INTERFACE IAction EXTENDS IObject

{attribute 'monitoring' := 'call'}
{attribute 'OPC.UA.DA.Property' := '1'}
{attribute 'OPC.UA.DA.Access' := '1'}
PROPERTY Busy : BOOL
GET
END_GET
END_PROPERTY

{attribute 'monitoring' := 'call'}
{attribute 'OPC.UA.DA.Property' := '1'}
{attribute 'OPC.UA.DA.Access' := '1'}
PROPERTY Done : BOOL
GET
END_GET
END_PROPERTY

{attribute 'monitoring' := 'call'}
{attribute 'OPC.UA.DA.Property' := '1'}
{attribute 'OPC.UA.DA.Access' := '1'}
PROPERTY Error : BOOL
GET
END_GET
END_PROPERTY

METHOD Execute
END_METHOD

END_INTERFACE

(* stored: Version 1.1.0.1
   Itf IAction: Id {33cd9918-3d9c-4cce-bc0c-72399b027fa3}
   Property Busy: Id {0bf76d8b-a1ea-4fc4-9149-9ac96039509d}
   Get Get: Id {bdaaed50-6e12-4f03-ab47-242eb0c00668}
   Property Done: Id {ef9f248d-3252-4ffa-aac3-0418e1335c37}
   Get Get: Id {dfaea843-6fb1-4dcb-81b1-47917a384f3e}
   Property Error: Id {7a16200e-ba54-400f-8eb2-30023de937d5}
   Get Get: Id {a77db7b9-68ef-4cc4-95b5-ec801cc3280a}
   Method Execute: Id {60763b55-6821-4e9a-af1a-388d0c4ba48c} *)
